PROGRAM MAIN
VAR
	a : UINT;
	b : UINT;
	c : UINT;
	x : UINT;
	y : UINT;
	i : UINT;
	j : UINT;
	k : UINT;
	q : UINT;
	w : UINT;
	e : UINT;
	
	
	
	bInit :	BOOL;
	
	bTRUE : BOOL;
END_VAR

a := a+1;
IF a = 10 THEN 
	FOR a := 1 TO 10 DO
		c := c + 1;
	END_FOR
END_IF

(*IF a = 10 THEN
	c := 0;
END_IF

FOR a := 1 TO 10 BY 1 DO
	c := c + 1;
END_FOR

CASE b OF
	1 :
	a := 1;
	2:
	b := 2;
	3:
	c := 3;
	4:
	a := 0;
	
END_CASE*)

END_PROGRAM

(* stored: Version 1.1.0.1, ProductVersion 3.1.4024.9
   POU MAIN: Id {e1db3390-2b00-4f43-8cf9-d9ba8703dbac}, SpecialFunc None *)
